// TIA Portal V16 export
// export: Created 2022-11-14T17:35:40.5139195Z, ExportSetting WithDefaults, DisplayName Totally Integrated Automation Portal, DisplayVersion V16, DisplayName TIA Portal Version Control Interface, DisplayVersion V16, DisplayName TIA Portal Openness, DisplayVersion V16, DisplayName STEP 7 Professional, DisplayVersion V16, DisplayName STEP 7 Safety, DisplayVersion V16, DisplayName WinCC Advanced, DisplayVersion V16
DATA_BLOCK "DB07_TopAux"   // DB7
{ S7_Optimized_Access := 'FALSE' }
AUTHOR : Robopac
VERSION : 0.0
// stored: AutoNumber false, IsOnlyStoredInLoadMemory false, IsWriteProtectedInAS false
   VAR RETAIN
      VB700 : Byte := 16#00;
      V701_0 : Bool := TRUE;   // Top film is wrapped
      V701_1 : Bool := FALSE;   // Support memory for top wrapped
      V701_2 : Bool := FALSE;
      V701_3 : Bool := FALSE;
      V701_4 : Bool := FALSE;
      V701_5 : Bool := FALSE;
      V701_6 : Bool := FALSE;
      V701_7 : Bool := FALSE;
   END_VAR
BEGIN
END_DATA_BLOCK
